// TIA Portal project "Test_2" (V17)

(* hardware
DEVICE "S7-1200 station_1"  S7-1200 Station
   slot 0: "Rack_0"  S7-1200 Rack  Rack  V1.0
   slot 1: "PLC_1"  CPU 1214C DC/DC/DC  6ES7 214-1AG40-0XB0  V4.4
   slot 3: "AQ 1x12BIT_1"  AQ1 signal board  6ES7 232-4HA30-0XB0  V1.0
   slot 101: "CM 1243-5"  CM 1243-5  6GK7 243-5DX30-0XE0  V1.3
*)

// ===== PLC "PLC_1"  CPU 1214C DC/DC/DC =====

VAR_GLOBAL   // PLC tag table "Default tag table"
   "Error_WWW" AT %MW200 : Int;
   "Wyjście_obroty" AT %QW80 : Word;
   "Wejścia_impulsy" AT %ID1000 : DWord;
   "Pamięć_impulsy" AT %MD1004 : DWord;
   "STATUS_HSC" AT %MW12 : Word;
   "Pamięć_alarmu" AT %M8.0 : Bool;
   "Stan_alarmu" AT %MW120 : Word;
   "Wyłącz_impulsy" AT %MW70 : Word;
END_VAR

DATA_BLOCK "WWW"   // DB1
{ S7_Optimized_Access := 'TRUE' }
VERSION : 0.1
   VAR
      Start : Bool;
      Stop : Bool;
      Zwiększ : Bool;
      Zmniejsz : Bool;
      Alarm_start : Bool;
      Potwierdzenie : Bool;
      impulsy : DWord;
   END_VAR
BEGIN
END_DATA_BLOCK

DATA_BLOCK "Obroty_DB"   // DB4
{ S7_Optimized_Access := 'TRUE' }
VERSION : 0.1
// stored: InstanceOfName Silnik DC | Kanał alarmowy
"Silnik DC | Kanał alarmowy"
BEGIN
END_DATA_BLOCK

// folder: System blocks/Program resources

DATA_BLOCK "IEC_Timer_0_DB_4"   // DB2
{ S7_Optimized_Access := 'TRUE' }
AUTHOR : Simatic
FAMILY : IEC
NAME : IEC_TMR
VERSION : 1.0
// stored: InstanceOfName IEC_TIMER
"IEC_TIMER"
BEGIN
END_DATA_BLOCK

DATA_BLOCK "IEC_Timer_0_DB"   // DB5
{ S7_Optimized_Access := 'TRUE' }
AUTHOR : Simatic
FAMILY : IEC
NAME : IEC_TMR
VERSION : 1.0
// stored: InstanceOfName IEC_TIMER
"IEC_TIMER"
BEGIN
END_DATA_BLOCK

DATA_BLOCK "IEC_Timer_0_DB_1"   // DB6
{ S7_Optimized_Access := 'TRUE' }
AUTHOR : Simatic
FAMILY : IEC
NAME : IEC_TMR
VERSION : 1.0
// stored: InstanceOfName IEC_TIMER
"IEC_TIMER"
BEGIN
END_DATA_BLOCK

DATA_BLOCK "IEC_Timer_0_DB_2"   // DB7
{ S7_Optimized_Access := 'TRUE' }
AUTHOR : Simatic
FAMILY : IEC
NAME : IEC_TMR
VERSION : 1.0
// stored: InstanceOfName IEC_TIMER
"IEC_TIMER"
BEGIN
END_DATA_BLOCK

DATA_BLOCK "IEC_Timer_0_DB_3"   // DB8
{ S7_Optimized_Access := 'TRUE' }
AUTHOR : Simatic
FAMILY : IEC
NAME : IEC_TMR
VERSION : 1.0
// stored: InstanceOfName IEC_TIMER
"IEC_TIMER"
BEGIN
END_DATA_BLOCK

DATA_BLOCK "IEC_Timer_0_DB_5"   // DB10
{ S7_Optimized_Access := 'TRUE' }
AUTHOR : Simatic
FAMILY : IEC
NAME : IEC_TMR
VERSION : 1.0
// stored: InstanceOfName IEC_TIMER
"IEC_TIMER"
BEGIN
END_DATA_BLOCK

// folder: (top level)

FUNCTION_BLOCK "Silnik DC | Kanał alarmowy"   // FB1, LAD
{ S7_Optimized_Access := 'TRUE' }
VERSION : 0.1
   VAR_OUTPUT
      alarm_stan : Word;
   END_VAR
   VAR_IN_OUT
      Start_WWW : Bool;
      Słowo_prędkość : Word;
      Zwiększ_prędkość_WWW : Bool;
      Zmniejsz_prędkość_WWW : Bool;
      Stop_WWW : Bool;
      Pam_Alarmu : Bool;
      Alarm_Start : Bool;
      Alarm_Potwierdzenie : Bool;
      Prędkość_zmienna : Word;
   END_VAR
   VAR_TEMP
      Zbocze_alarm : Bool;
   END_VAR
   VAR_TEMP   // added for the SCL form of the ladder/FBD networks
      _w1 : Bool;
      _w2 : Bool;
   END_VAR
BEGIN

REGION Network 1: Przycisk Start
   // Ustawienie wartości zmiennej słowo_prędkość na 5000
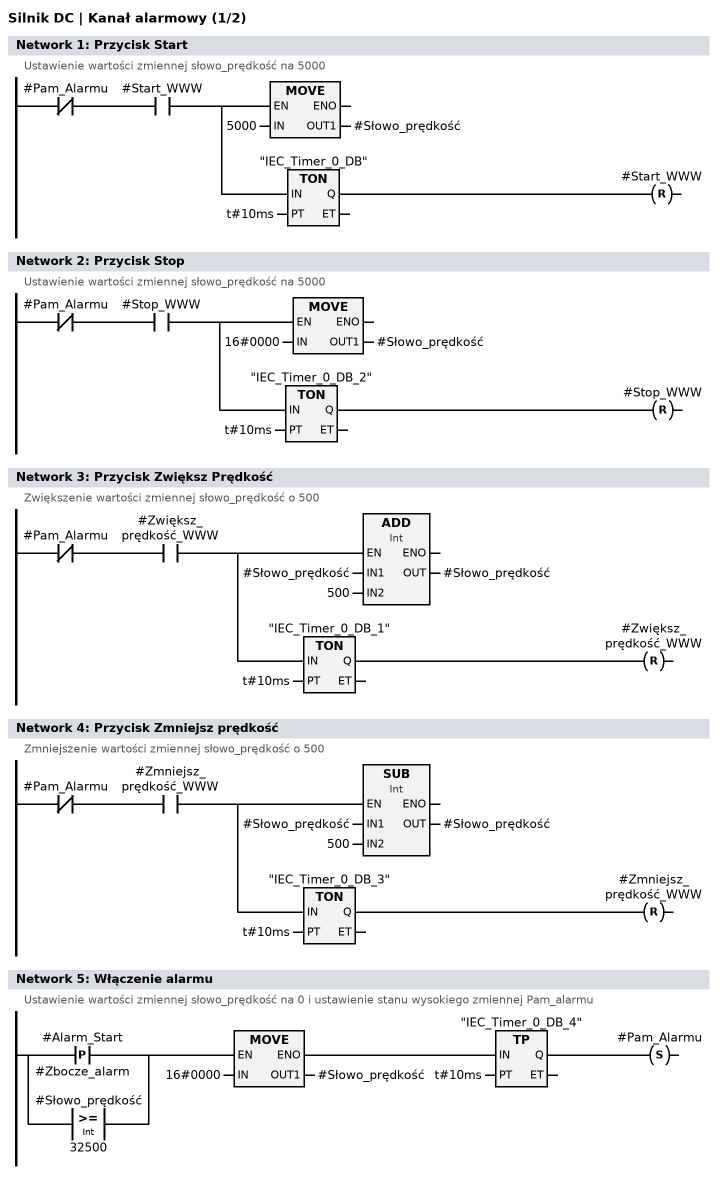
   #_w1 := NOT #Pam_Alarmu AND #Start_WWW;
   IF #_w1 THEN #Słowo_prędkość := 5000; END_IF;
   "IEC_Timer_0_DB".TON(IN := #_w1, PT := t#10ms);
   IF "IEC_Timer_0_DB".Q THEN #Start_WWW := FALSE; END_IF;
END_REGION

REGION Network 2: Przycisk Stop
   // Ustawienie wartości zmiennej słowo_prędkość na 5000
   #_w1 := NOT #Pam_Alarmu AND #Stop_WWW;
   IF #_w1 THEN #Słowo_prędkość := 16#0000; END_IF;
   "IEC_Timer_0_DB_2".TON(IN := #_w1, PT := t#10ms);
   IF "IEC_Timer_0_DB_2".Q THEN #Stop_WWW := FALSE; END_IF;
END_REGION

REGION Network 3: Przycisk Zwiększ Prędkość
   // Zwiększenie wartości zmiennej słowo_prędkość o 500
   #_w1 := NOT #Pam_Alarmu AND #Zwiększ_prędkość_WWW;
   IF #_w1 THEN #Słowo_prędkość := #Słowo_prędkość + 500; END_IF;
   "IEC_Timer_0_DB_1".TON(IN := #_w1, PT := t#10ms);
   IF "IEC_Timer_0_DB_1".Q THEN #Zwiększ_prędkość_WWW := FALSE; END_IF;
END_REGION

REGION Network 4: Przycisk Zmniejsz prędkość
   // Zmniejszenie wartości zmiennej słowo_prędkość o 500
   #_w1 := NOT #Pam_Alarmu AND #Zmniejsz_prędkość_WWW;
   IF #_w1 THEN #Słowo_prędkość := #Słowo_prędkość - 500; END_IF;
   "IEC_Timer_0_DB_3".TON(IN := #_w1, PT := t#10ms);
   IF "IEC_Timer_0_DB_3".Q THEN #Zmniejsz_prędkość_WWW := FALSE; END_IF;
END_REGION

REGION Network 5: Włączenie alarmu
   // Ustawienie wartości zmiennej słowo_prędkość na 0 i ustawienie stanu wysokiego zmiennej Pam_alarmu
   #_w1 := #Alarm_Start AND NOT #Zbocze_alarm;   // rising edge of #Alarm_Start
   #Zbocze_alarm := #Alarm_Start;
   #_w2 := #_w1 OR (#Słowo_prędkość >= 32500);
   IF #_w2 THEN #Słowo_prędkość := 16#0000; END_IF;
   "IEC_Timer_0_DB_4".TP(IN := #_w2, PT := t#10ms);
   IF "IEC_Timer_0_DB_4".Q THEN #Pam_Alarmu := TRUE; END_IF;
END_REGION

REGION Network 6: Potwierdzenie alarmu
   // Zmiana stanu zmiennej Pam_alarmu na stan niski
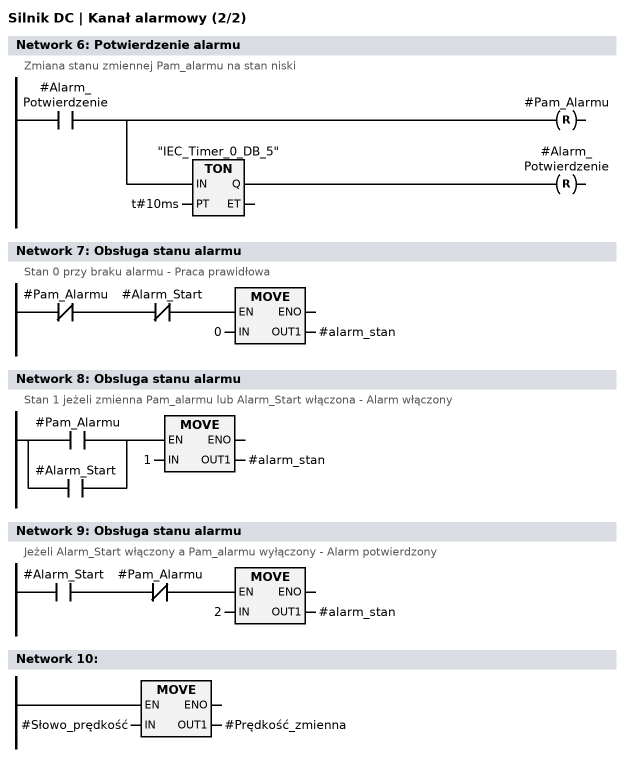
   IF #Alarm_Potwierdzenie THEN #Pam_Alarmu := FALSE; END_IF;
   "IEC_Timer_0_DB_5".TON(IN := #Alarm_Potwierdzenie, PT := t#10ms);
   IF "IEC_Timer_0_DB_5".Q THEN #Alarm_Potwierdzenie := FALSE; END_IF;
END_REGION

REGION Network 7: Obsługa stanu alarmu
   // Stan 0 przy braku alarmu - Praca prawidłowa
   RUNG wire#powerrail
      I_Contact( #Pam_Alarmu )
      I_Contact( #Alarm_Start )
      Move(in := 0, out1 => #alarm_stan)
   END_RUNG
   // the same network as SCL:
   IF NOT #Pam_Alarmu AND NOT #Alarm_Start THEN #alarm_stan := 0; END_IF;
END_REGION

REGION Network 8: Obsluga stanu alarmu
   // Stan 1 jeżeli zmienna Pam_alarmu lub Alarm_Start włączona - Alarm włączony
   RUNG wire#powerrail
      Contact( #Pam_Alarmu )
      wire#w1
      Move(in := 1, out1 => #alarm_stan)
   END_RUNG
   RUNG wire#powerrail
      Contact( #Alarm_Start )
   END_RUNG wire#w1
   // the same network as SCL:
   IF #Pam_Alarmu OR #Alarm_Start THEN #alarm_stan := 1; END_IF;
END_REGION

REGION Network 9: Obsługa stanu alarmu
   // Jeżeli Alarm_Start włączony a Pam_alarmu wyłączony - Alarm potwierdzony
   RUNG wire#powerrail
      Contact( #Alarm_Start )
      I_Contact( #Pam_Alarmu )
      Move(in := 2, out1 => #alarm_stan)
   END_RUNG
   // the same network as SCL:
   IF #Alarm_Start AND NOT #Pam_Alarmu THEN #alarm_stan := 2; END_IF;
END_REGION

REGION Network 10
   RUNG wire#powerrail
      Move(in := #Słowo_prędkość, out1 => #Prędkość_zmienna)
   END_RUNG
   // the same network as SCL:
   #Prędkość_zmienna := #Słowo_prędkość;
END_REGION
END_FUNCTION_BLOCK

ORGANIZATION_BLOCK "Main"   // OB1, LAD, ProgramCycle
TITLE = "Main Program Sweep (Cycle)"
{ S7_Optimized_Access := 'TRUE' }
VERSION : 0.1
   VAR_INPUT
      Initial_Call : Bool;   // Initial call of this OB
      Remanence : Bool;   // =True, if remanent data are available
   END_VAR
BEGIN

REGION Network 1: Inicjalizacja / synchronizacja strony
   // CTRL_DB: Data block ze stroną| RET_VAL: Informacja o błędach
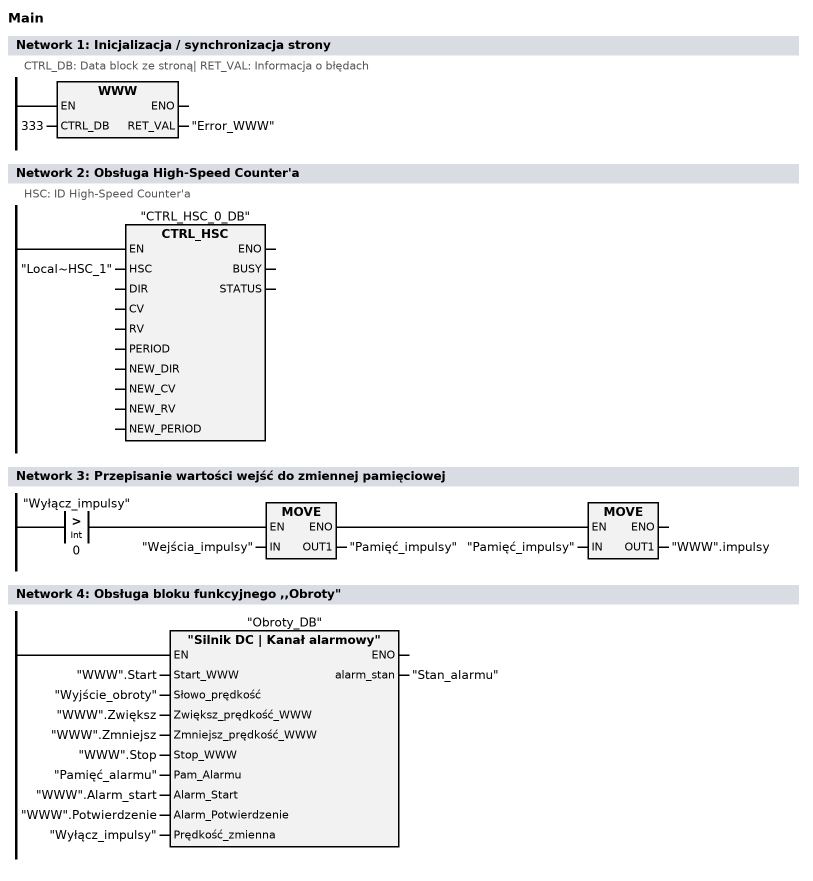
   "Error_WWW" := WWW(CTRL_DB := 333);
END_REGION

REGION Network 2: Obsługa High-Speed Counter'a
   // HSC: ID High-Speed Counter'a
   "CTRL_HSC_0_DB"(HSC := "Local~HSC_1");   // CTRL_HSC
END_REGION

REGION Network 3: Przepisanie wartości wejść do zmiennej pamięciowej
   RUNG wire#powerrail
      { S7_Templates := "SrcType := Int" } GT_Contact(in1 := "Wyłącz_impulsy", in2 := 0)
      Move(in := "Wejścia_impulsy", out1 => "Pamięć_impulsy")
      Move(in := "Pamięć_impulsy", out1 => "WWW".impulsy)
   END_RUNG
   // the same network as SCL:
   IF "Wyłącz_impulsy" > 0 THEN
       "Pamięć_impulsy" := "Wejścia_impulsy";
       "WWW".impulsy := "Pamięć_impulsy";
   END_IF;
END_REGION

REGION Network 4: Obsługa bloku funkcyjnego ,,Obroty"
   RUNG wire#powerrail
      "Obroty_DB"(Start_WWW := "WWW".Start, Słowo_prędkość := "Wyjście_obroty", Zwiększ_prędkość_WWW := "WWW".Zwiększ, Zmniejsz_prędkość_WWW := "WWW".Zmniejsz, Stop_WWW := "WWW".Stop, Pam_Alarmu := "Pamięć_alarmu", Alarm_Start := "WWW".Alarm_start, Alarm_Potwierdzenie := "WWW".Potwierdzenie, Prędkość_zmienna := "Wyłącz_impulsy", alarm_stan => "Stan_alarmu")
   END_RUNG
   // the same network as SCL:
   "Obroty_DB"(Start_WWW := "WWW".Start,   // "Silnik DC | Kanał alarmowy"
               Słowo_prędkość := "Wyjście_obroty",
               Zwiększ_prędkość_WWW := "WWW".Zwiększ,
               Zmniejsz_prędkość_WWW := "WWW".Zmniejsz,
               Stop_WWW := "WWW".Stop,
               Pam_Alarmu := "Pamięć_alarmu",
               Alarm_Start := "WWW".Alarm_start,
               Alarm_Potwierdzenie := "WWW".Potwierdzenie,
               Prędkość_zmienna := "Wyłącz_impulsy",
               alarm_stan => "Stan_alarmu");
END_REGION
END_ORGANIZATION_BLOCK